PROGRAM MAIN
VAR
END_VAR

END_PROGRAM

(* stored: Version 1.1.0.1
   POU MAIN: Id {2a11b0b8-4c62-4315-92a5-302ee14477bd} *)
